// Mitsubishi GX Developer project: 12-1105培林與軸套自動壓合機   PLC: FX1N

PROGRAM MAIN
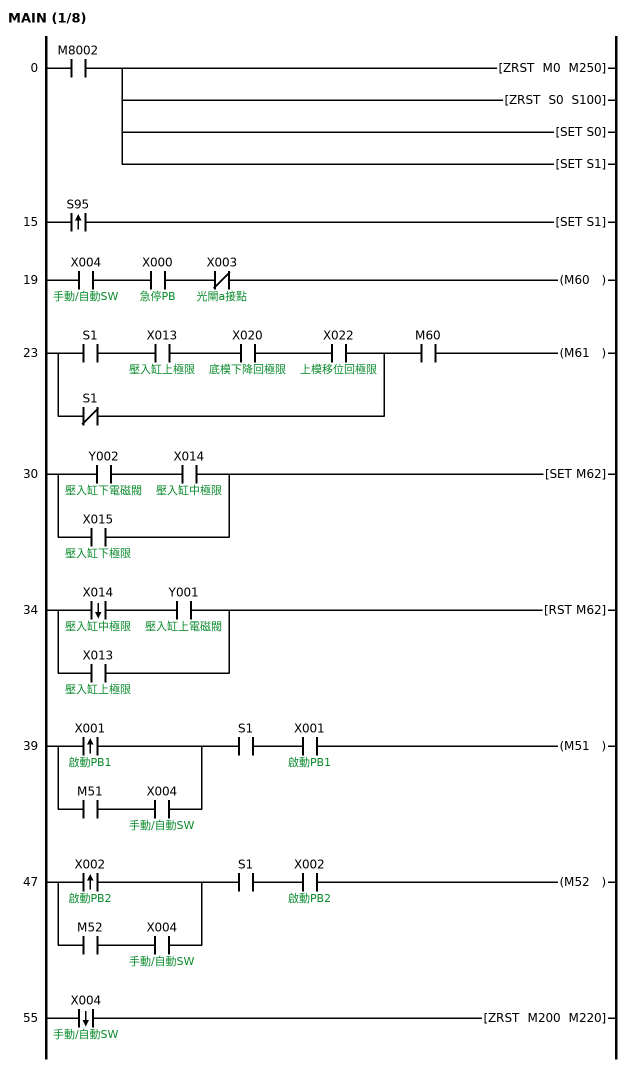
0     LD      M8002
      ZRST    M0 M250
      ZRST    S0 S100
      SET     S0
      SET     S1
15    LDP     S95
      SET     S1
19    LD      X004  ; 手動/自動SW
      AND     X000  ; 急停PB
      ANI     X003  ; 光閘a接點
      OUT     M60
23    LD      S1
      AND     X013  ; 壓入缸上極限
      AND     X020  ; 底模下降回極限
      AND     X022  ; 上模移位回極限
      ORI     S1
      AND     M60
      OUT     M61
30    LD      Y002  ; 壓入缸下電磁閥
      AND     X014  ; 壓入缸中極限
      OR      X015  ; 壓入缸下極限
      SET     M62
34    LDF     X014  ; 壓入缸中極限
      AND     Y001  ; 壓入缸上電磁閥
      OR      X013  ; 壓入缸上極限
      RST     M62
39    LDP     X001  ; 啟動PB1
      LD      M51
      AND     X004  ; 手動/自動SW
      ORB
      AND     S1
      AND     X001  ; 啟動PB1
      OUT     M51
47    LDP     X002  ; 啟動PB2
      LD      M52
      AND     X004  ; 手動/自動SW
      ORB
      AND     S1
      AND     X002  ; 啟動PB2
      OUT     M52
55    LDF     X004  ; 手動/自動SW
      ZRST    M200 M220
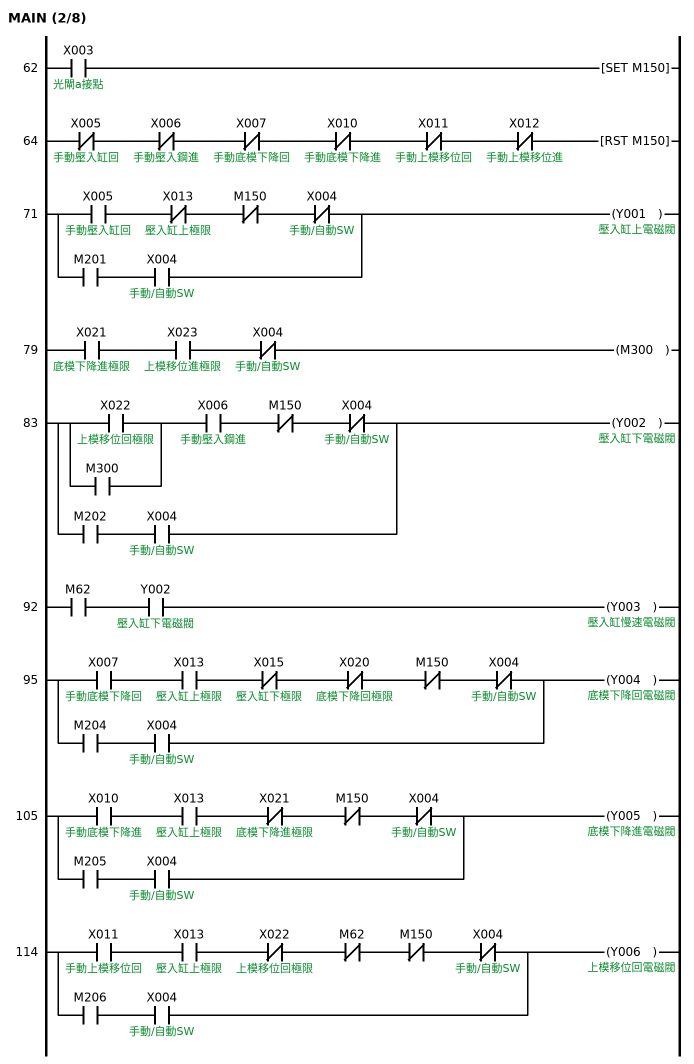
62    LD      X003  ; 光閘a接點
      SET     M150
64    LDI     X005  ; 手動壓入缸回
      ANI     X006  ; 手動壓入鋼進
      ANI     X007  ; 手動底模下降回
      ANI     X010  ; 手動底模下降進
      ANI     X011  ; 手動上模移位回
      ANI     X012  ; 手動上模移位進
      RST     M150
71    LD      X005  ; 手動壓入缸回
      ANI     X013  ; 壓入缸上極限
      ANI     M150
      ANI     X004  ; 手動/自動SW
      LD      M201
      AND     X004  ; 手動/自動SW
      ORB
      OUT     Y001  ; 壓入缸上電磁閥
79    LD      X021  ; 底模下降進極限
      AND     X023  ; 上模移位進極限
      ANI     X004  ; 手動/自動SW
      OUT     M300
83    LD      X022  ; 上模移位回極限
      OR      M300
      AND     X006  ; 手動壓入鋼進
      ANI     M150
      ANI     X004  ; 手動/自動SW
      LD      M202
      AND     X004  ; 手動/自動SW
      ORB
      OUT     Y002  ; 壓入缸下電磁閥
92    LD      M62
      AND     Y002  ; 壓入缸下電磁閥
      OUT     Y003  ; 壓入缸慢速電磁閥
95    LD      X007  ; 手動底模下降回
      AND     X013  ; 壓入缸上極限
      ANI     X015  ; 壓入缸下極限
      ANI     X020  ; 底模下降回極限
      ANI     M150
      ANI     X004  ; 手動/自動SW
      LD      M204
      AND     X004  ; 手動/自動SW
      ORB
      OUT     Y004  ; 底模下降回電磁閥
105   LD      X010  ; 手動底模下降進
      AND     X013  ; 壓入缸上極限
      ANI     X021  ; 底模下降進極限
      ANI     M150
      ANI     X004  ; 手動/自動SW
      LD      M205
      AND     X004  ; 手動/自動SW
      ORB
      OUT     Y005  ; 底模下降進電磁閥
114   LD      X011  ; 手動上模移位回
      AND     X013  ; 壓入缸上極限
      ANI     X022  ; 上模移位回極限
      ANI     M62
      ANI     M150
      ANI     X004  ; 手動/自動SW
      LD      M206
      AND     X004  ; 手動/自動SW
      ORB
      OUT     Y006  ; 上模移位回電磁閥
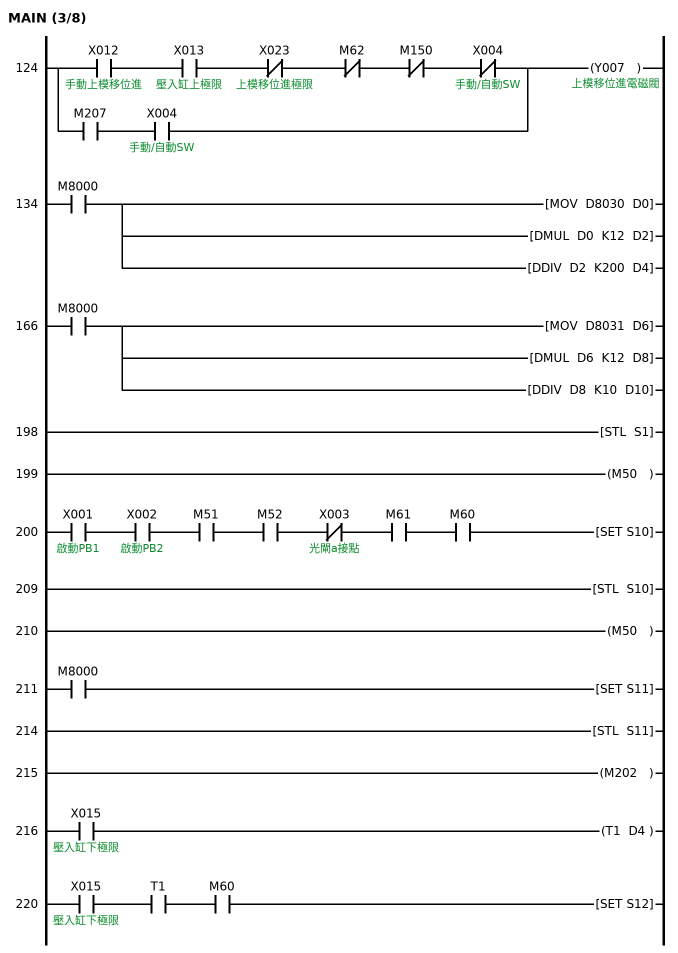
124   LD      X012  ; 手動上模移位進
      AND     X013  ; 壓入缸上極限
      ANI     X023  ; 上模移位進極限
      ANI     M62
      ANI     M150
      ANI     X004  ; 手動/自動SW
      LD      M207
      AND     X004  ; 手動/自動SW
      ORB
      OUT     Y007  ; 上模移位進電磁閥
134   LD      M8000
      MOV     D8030 D0
      DMUL    D0 K12 D2
      DDIV    D2 K200 D4
166   LD      M8000
      MOV     D8031 D6
      DMUL    D6 K12 D8
      DDIV    D8 K10 D10
198   STL     S1
199   OUT     M50
200   LD      X001  ; 啟動PB1
      AND     X002  ; 啟動PB2
      AND     M51
      AND     M52
      ANI     X003  ; 光閘a接點
      AND     M61
      AND     M60
      SET     S10
209   STL     S10
210   OUT     M50
211   LD      M8000
      SET     S11
214   STL     S11
215   OUT     M202
216   LD      X015  ; 壓入缸下極限
      OUT     T1 D4
220   LD      X015  ; 壓入缸下極限
      AND     T1
      AND     M60
      SET     S12
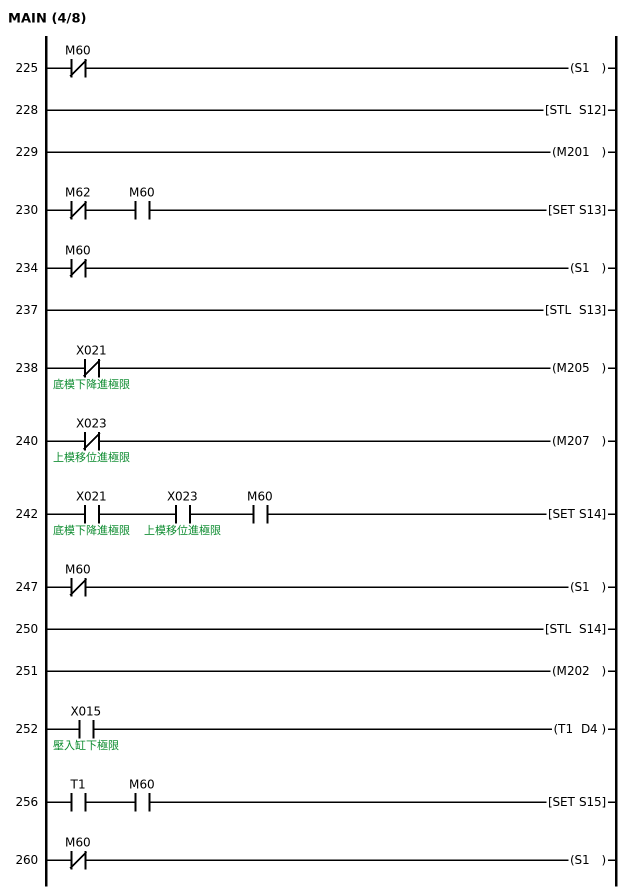
225   LDI     M60
      OUT     S1
228   STL     S12
229   OUT     M201
230   LDI     M62
      AND     M60
      SET     S13
234   LDI     M60
      OUT     S1
237   STL     S13
238   LDI     X021  ; 底模下降進極限
      OUT     M205
240   LDI     X023  ; 上模移位進極限
      OUT     M207
242   LD      X021  ; 底模下降進極限
      AND     X023  ; 上模移位進極限
      AND     M60
      SET     S14
247   LDI     M60
      OUT     S1
250   STL     S14
251   OUT     M202
252   LD      X015  ; 壓入缸下極限
      OUT     T1 D4
256   LD      T1
      AND     M60
      SET     S15
260   LDI     M60
      OUT     S1
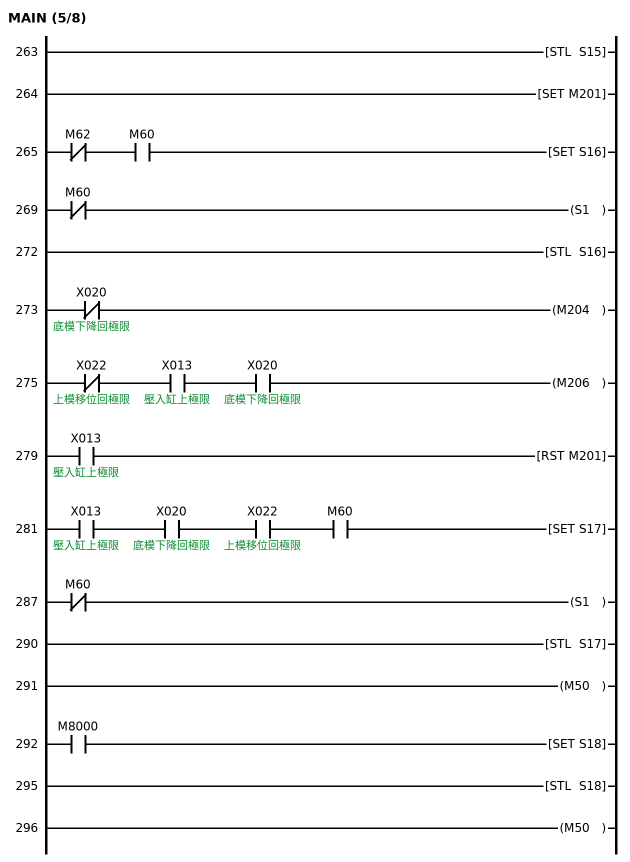
263   STL     S15
264   SET     M201
265   LDI     M62
      AND     M60
      SET     S16
269   LDI     M60
      OUT     S1
272   STL     S16
273   LDI     X020  ; 底模下降回極限
      OUT     M204
275   LDI     X022  ; 上模移位回極限
      AND     X013  ; 壓入缸上極限
      AND     X020  ; 底模下降回極限
      OUT     M206
279   LD      X013  ; 壓入缸上極限
      RST     M201
281   LD      X013  ; 壓入缸上極限
      AND     X020  ; 底模下降回極限
      AND     X022  ; 上模移位回極限
      AND     M60
      SET     S17
287   LDI     M60
      OUT     S1
290   STL     S17
291   OUT     M50
292   LD      M8000
      SET     S18
295   STL     S18
296   OUT     M50
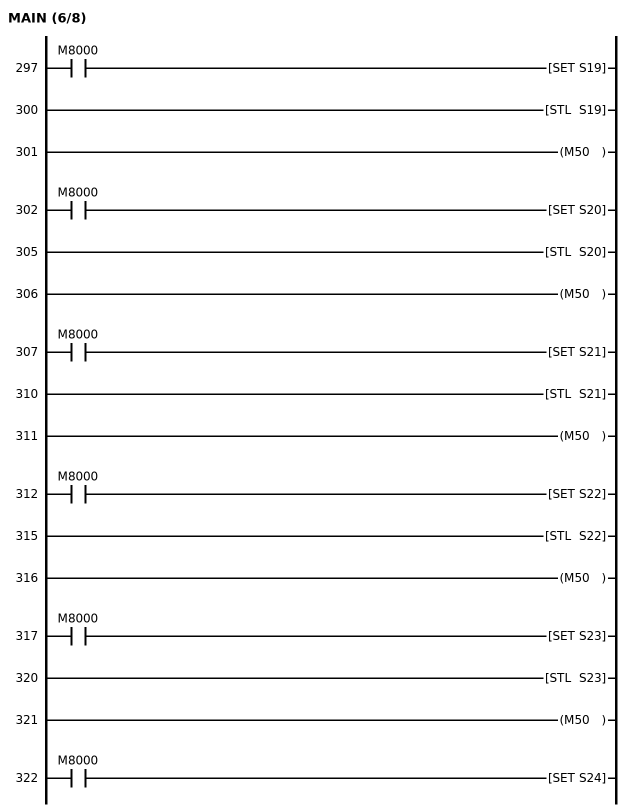
297   LD      M8000
      SET     S19
300   STL     S19
301   OUT     M50
302   LD      M8000
      SET     S20
305   STL     S20
306   OUT     M50
307   LD      M8000
      SET     S21
310   STL     S21
311   OUT     M50
312   LD      M8000
      SET     S22
315   STL     S22
316   OUT     M50
317   LD      M8000
      SET     S23
320   STL     S23
321   OUT     M50
322   LD      M8000
      SET     S24
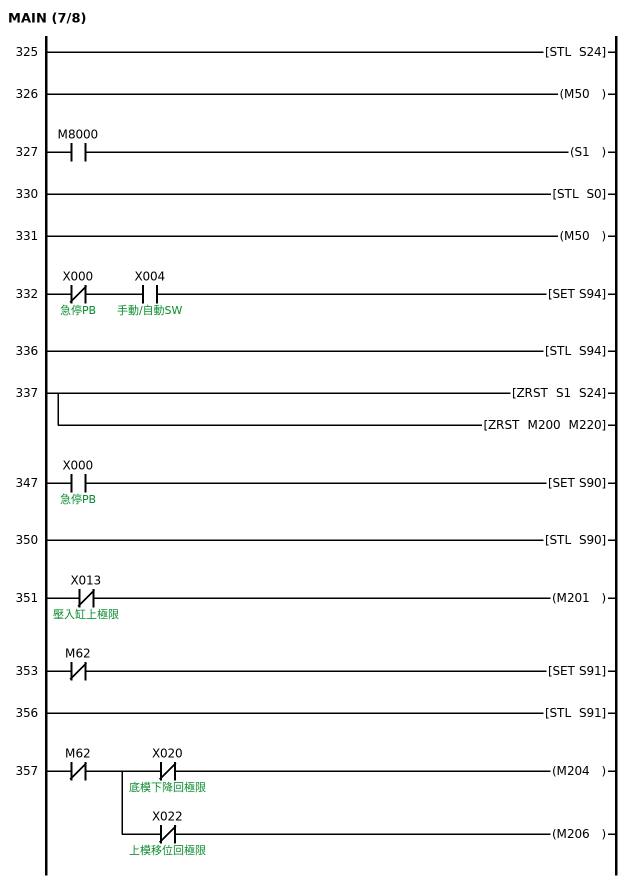
325   STL     S24
326   OUT     M50
327   LD      M8000
      OUT     S1
330   STL     S0
331   OUT     M50
332   LDI     X000  ; 急停PB
      AND     X004  ; 手動/自動SW
      SET     S94
336   STL     S94
337   ZRST    S1 S24
      ZRST    M200 M220
347   LD      X000  ; 急停PB
      SET     S90
350   STL     S90
351   LDI     X013  ; 壓入缸上極限
      OUT     M201
353   LDI     M62
      SET     S91
356   STL     S91
357   LDI     M62
      MPS
      ANI     X020  ; 底模下降回極限
      OUT     M204
      MPP
      ANI     X022  ; 上模移位回極限
      OUT     M206
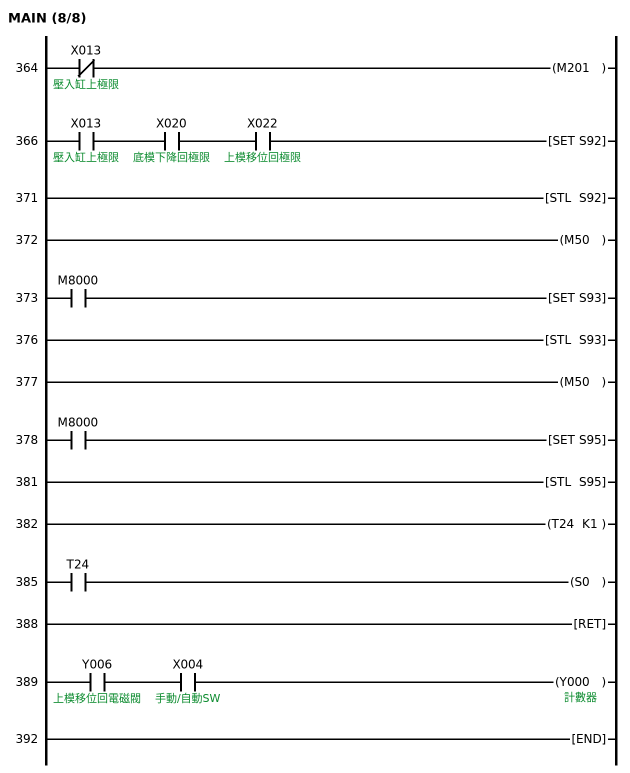
364   LDI     X013  ; 壓入缸上極限
      OUT     M201
366   LD      X013  ; 壓入缸上極限
      AND     X020  ; 底模下降回極限
      AND     X022  ; 上模移位回極限
      SET     S92
371   STL     S92
372   OUT     M50
373   LD      M8000
      SET     S93
376   STL     S93
377   OUT     M50
378   LD      M8000
      SET     S95
381   STL     S95
382   OUT     T24 K1
385   LD      T24
      OUT     S0
388   RET
389   LD      Y006  ; 上模移位回電磁閥
      AND     X004  ; 手動/自動SW
      OUT     Y000  ; 計數器
392   END
END_PROGRAM

// device comments not shown above
BL0  ; main
BL1  ; 直向順序
BL2  ; ALARM RESET(放在最後)
